// Mitsubishi GX Works2 project: part1 - Copy   PLC: FX3G

// global labels: Global1
VAR_GLOBAL
  start AT X007 : BOOL;
  helpStart AT M0 : BOOL;
  end_day AT X010 : BOOL;
  help_light AT M1 : BOOL;
  TC_200 AT TC200 : BOOL;
END_VAR
VAR_GLOBAL CONSTANT
  TIMER_1 : INT := 300;
END_VAR
VAR_GLOBAL
  TS_200 AT TS200 : BOOL;
  help_light2 AT M2 : BOOL;
  if_enough_stock AT M3 : BOOL;
  day_off AT M4 : BOOL;
END_VAR
VAR_GLOBAL CONSTANT
  zero : INT;
END_VAR
VAR_GLOBAL
  Cream AT D1100 : INT;
  cream_stock : INT;
  Chocolate AT D1101 : INT;
  chocolate_stock AT D1102 : INT;
  biscuit AT D1103 : INT;
  biscuit_stock AT D1104 : INT;
  start_Ziluf AT X011 : BOOL;
END_VAR
VAR_GLOBAL CONSTANT
  Cream300 : INT := 300;
END_VAR
VAR_GLOBAL
  ziluf_container AT D1105 : INT;
END_VAR
VAR_GLOBAL CONSTANT
  biscuit6 : INT := 6;
END_VAR
VAR_GLOBAL
  machineA AT X010 : BOOL;
  sen_mishtah AT X001 : BOOL;
  sen_camera AT X002 : BOOL;
  stop_machineA AT X005 : BOOL;
  sen_temp30 AT X003 : BOOL;
  sen_temp15 AT X004 : BOOL;
  ziluf_on AT Y004 : BOOL;
  finish_ziluf AT Y000 : BOOL;
  start_day AT Y007 : BOOL;
  m_5 AT M5 : BOOL;
  m_6 AT M6 : BOOL;
  m_7 AT M7 : BOOL;
  y_0 AT Y000 : BOOL;
  y_1 AT Y001 : BOOL;
  TS_1 AT TS1 : BOOL;
  m_0 AT M0 : BOOL;
  m_8 AT M8 : BOOL;
  TC_1 AT TC1 : BOOL;
END_VAR
VAR_GLOBAL CONSTANT
  sec_40 : INT := 40;
END_VAR
VAR_GLOBAL
  TC_2 AT TC2 : BOOL;
END_VAR
VAR_GLOBAL CONSTANT
  sec_1 : INT := 10;
END_VAR
VAR_GLOBAL
  TS_2 AT TS2 : BOOL;
  TC_3 AT TC3 : BOOL;
  TS_3 AT TS3 : BOOL;
  start_machineB AT X006 : BOOL;
END_VAR
VAR_GLOBAL CONSTANT
  div_400 : INT := 400;
END_VAR
VAR_GLOBAL
  analog_value : INT;
  m_9 AT M9 : BOOL;
END_VAR
VAR_GLOBAL CONSTANT
  Con : INT;
  Con0 : INT := 5;
  Con5 : INT := 5;
  CoN10 : INT := 10;
END_VAR
VAR_GLOBAL
  double_top AT M10 : BOOL;
END_VAR
VAR_GLOBAL CONSTANT
  Con6 : INT := 6;
END_VAR
VAR_GLOBAL
  regular_top AT M11 : BOOL;
  outRange AT M12 : BOOL;
  dip_container AT D1106 : INT;
END_VAR
VAR_GLOBAL CONSTANT
  Chocloate120 : INT := 120;
  Chocloate240 : INT := 240;
END_VAR
VAR_GLOBAL
  TC_4 AT TC4 : BOOL;
END_VAR
VAR_GLOBAL CONSTANT
  sec5 : INT := 50;
END_VAR
VAR_GLOBAL
  end_dip AT Y003 : BOOL;
  analog_input1 AT D8280 : INT;
  Analogvalue_result : BOOL;
  GT_result : REAL;
  TC_5 AT TC5 : BOOL;
END_VAR
VAR_GLOBAL CONSTANT
  sec_4 : INT := 40;
END_VAR
VAR_GLOBAL
  TS_5 AT TS5 : BOOL;
  y_3 AT Y003 : BOOL;
  finish_top AT M13 : BOOL;
  finish_regulartop AT M13 : BOOL;
  finish_doubletop AT M14 : BOOL;
  start_ariza AT X000 : BOOL;
  CC_1 AT CC1 : BOOL;
END_VAR
VAR_GLOBAL CONSTANT
  X0_value5 : INT := 5;
END_VAR
VAR_GLOBAL
  sof_ariza : BOOL;
  ariza AT X000 : BOOL;
  CC_2 AT CC2 : BOOL;
END_VAR
VAR_GLOBAL CONSTANT
  X0_value6 : INT := 6;
END_VAR
VAR_GLOBAL
  CS_1 AT CS1 : BOOL;
  CS_2 AT CS2 : BOOL;
  y_2 AT Y002 : BOOL;
  machineAhelp AT M15 : BOOL;
  end_prep AT M16 : BOOL;
  finish_prep AT M16 : BOOL;
  finish_iteration AT M17 : BOOL;
END_VAR
VAR_GLOBAL CONSTANT
  amount_6 : INT := 6;
END_VAR
VAR_GLOBAL
  total_krembo : INT;
  Check_stock AT M18 : BOOL;
END_VAR
VAR_GLOBAL CONSTANT
  min_6 : INT;
  min_300 : INT := 300;
  min_240 : INT := 240;
END_VAR
VAR_GLOBAL
  analog_output AT D8282 : INT;
END_VAR
VAR_GLOBAL CONSTANT
  Con_40 : INT := 40;
END_VAR
VAR_GLOBAL
  output_value : INT;
  if_enough_buiscit AT M19 : BOOL;
  if_enough_cream AT M20 : BOOL;
  if_enough_chocolate AT M21 : BOOL;
  TC_6 AT TC6 : BOOL;
  M_22 AT M22 : BOOL;
  TS_6 AT TS6 : BOOL;
END_VAR
VAR_GLOBAL CONSTANT
  sec_05 : INT := 5;
END_VAR
VAR_GLOBAL
  TC_7 AT TC7 : BOOL;
  TS_7 AT TS7 : BOOL;
  stock_ok AT M23 : BOOL;
  Check_first_stock AT M24 : BOOL;
  finish_fillstock AT M25 : BOOL;
  TC_8 AT TC8 : BOOL;
  TS_8 AT TS8 : BOOL;
END_VAR
VAR_GLOBAL CONSTANT
  CoNST0 : INT;
END_VAR
VAR_GLOBAL
  help_start AT M27 : BOOL;
  toping_kind : INT;
END_VAR

// task Task_01 (event TRUE, interval 0, priority 31): POU_01

PROGRAM POU_01
(* structured ladder/FBD written out as ST: instructions are called as NAME(EN, inputs, outputs); _pN, _eN, _tN stand for wires *)
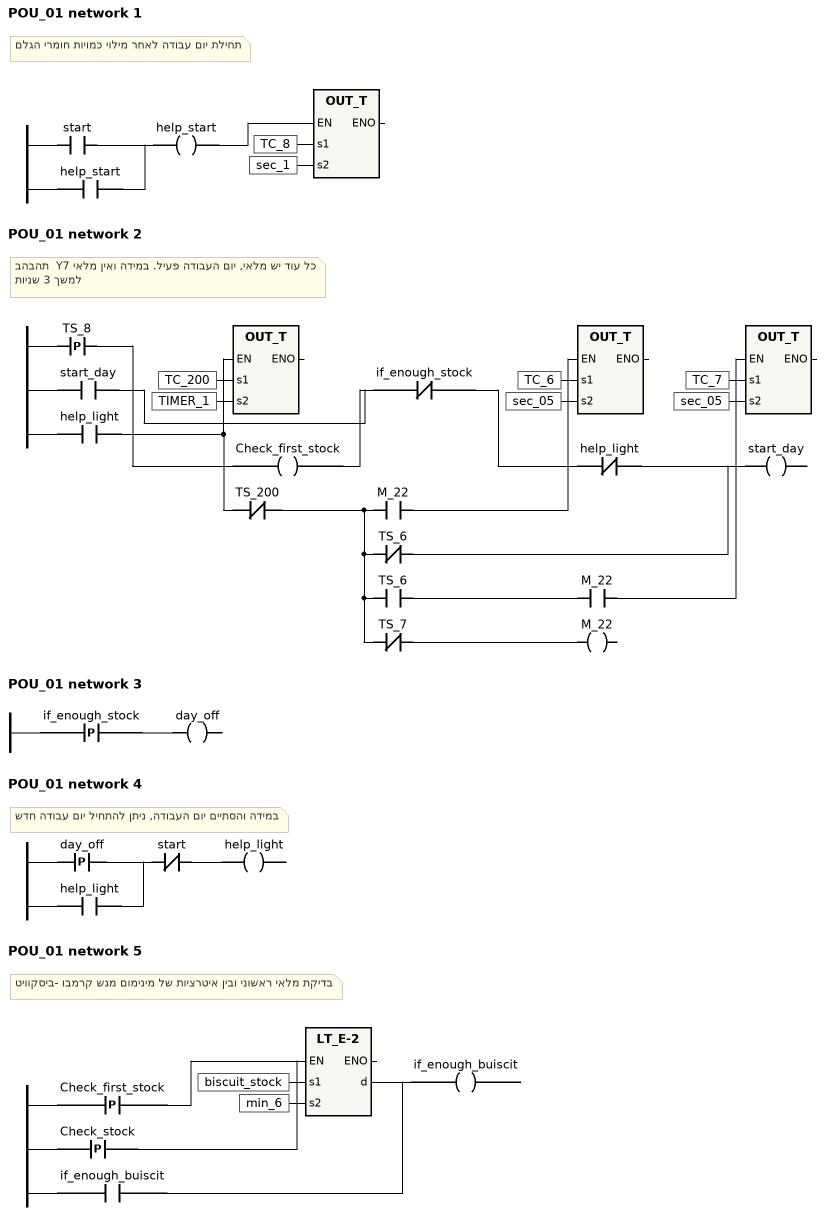
(* network 1 *)
(* תחילת יום עבודה לאחר מילוי כמויות חומרי הגלם *)
_p1 := start OR help_start;
help_start := _p1;
OUT_T(_p1, TC_8, sec_1);
(* network 2 *)
(* כל עוד יש מלאי, יום העבודה פעיל. במידה ואין מלאי Y7  תהבהב למשך 3 שניות *)
_p1 := LDP(TRUE, TS_8);
Check_first_stock := _p1;
_p2 := help_light AND NOT TS_200;
start_day := (((_p1 OR start_day) AND NOT if_enough_stock) AND NOT help_light) OR (_p2 AND NOT TS_6);
OUT_T(help_light, TC_200, TIMER_1);
OUT_T(_p2 AND M_22, TC_6, sec_05);
OUT_T(_p2 AND TS_6 AND M_22, TC_7, sec_05);
M_22 := _p2 AND NOT TS_7;
(* network 3 *)
day_off := LDP(TRUE, if_enough_stock);
(* network 4 *)
(* במידה והסתיים יום העבודה, ניתן להתחיל יום עבודה חדש *)
help_light := (LDP(TRUE, day_off) OR help_light) AND NOT start;
(* network 5 *)
(* בדיקת מלאי ראשוני ובין איטרציות של מינימום מגש קרמבו -ביסקוויט *)
LT_E(LDP(TRUE, Check_first_stock) OR LDP(TRUE, Check_stock), biscuit_stock, min_6, _t1);
if_enough_buiscit := _t1 OR if_enough_buiscit;
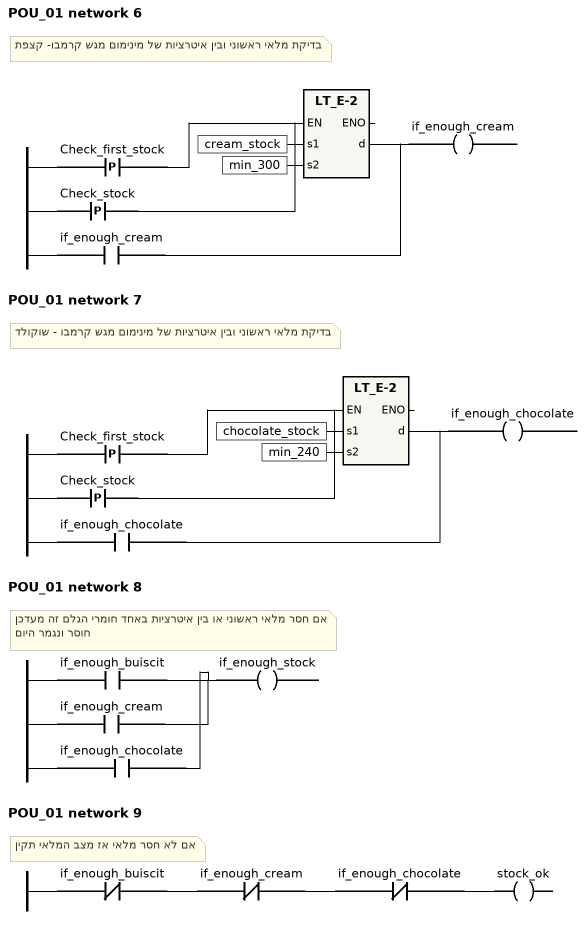
(* network 6 *)
(* בדיקת מלאי ראשוני ובין איטרציות של מינימום מגש קרמבו- קצפת *)
LT_E(LDP(TRUE, Check_first_stock) OR LDP(TRUE, Check_stock), cream_stock, min_300, _t1);
if_enough_cream := _t1 OR if_enough_cream;
(* network 7 *)
(* בדיקת מלאי ראשוני ובין איטרציות של מינימום מגש קרמבו - שוקולד *)
LT_E(LDP(TRUE, Check_first_stock) OR LDP(TRUE, Check_stock), chocolate_stock, min_240, _t1);
if_enough_chocolate := _t1 OR if_enough_chocolate;
(* network 8 *)
(* אם חסר מלאי ראשוני או בין איטרציות באחד חומרי הגלם זה מעדכן חוסר ונגמר היום *)
if_enough_stock := if_enough_buiscit OR if_enough_cream OR if_enough_chocolate;
(* network 9 *)
(* אם לא חסר מלאי אז מצב המלאי תקין *)
stock_ok := NOT if_enough_buiscit AND NOT if_enough_cream AND NOT if_enough_chocolate;
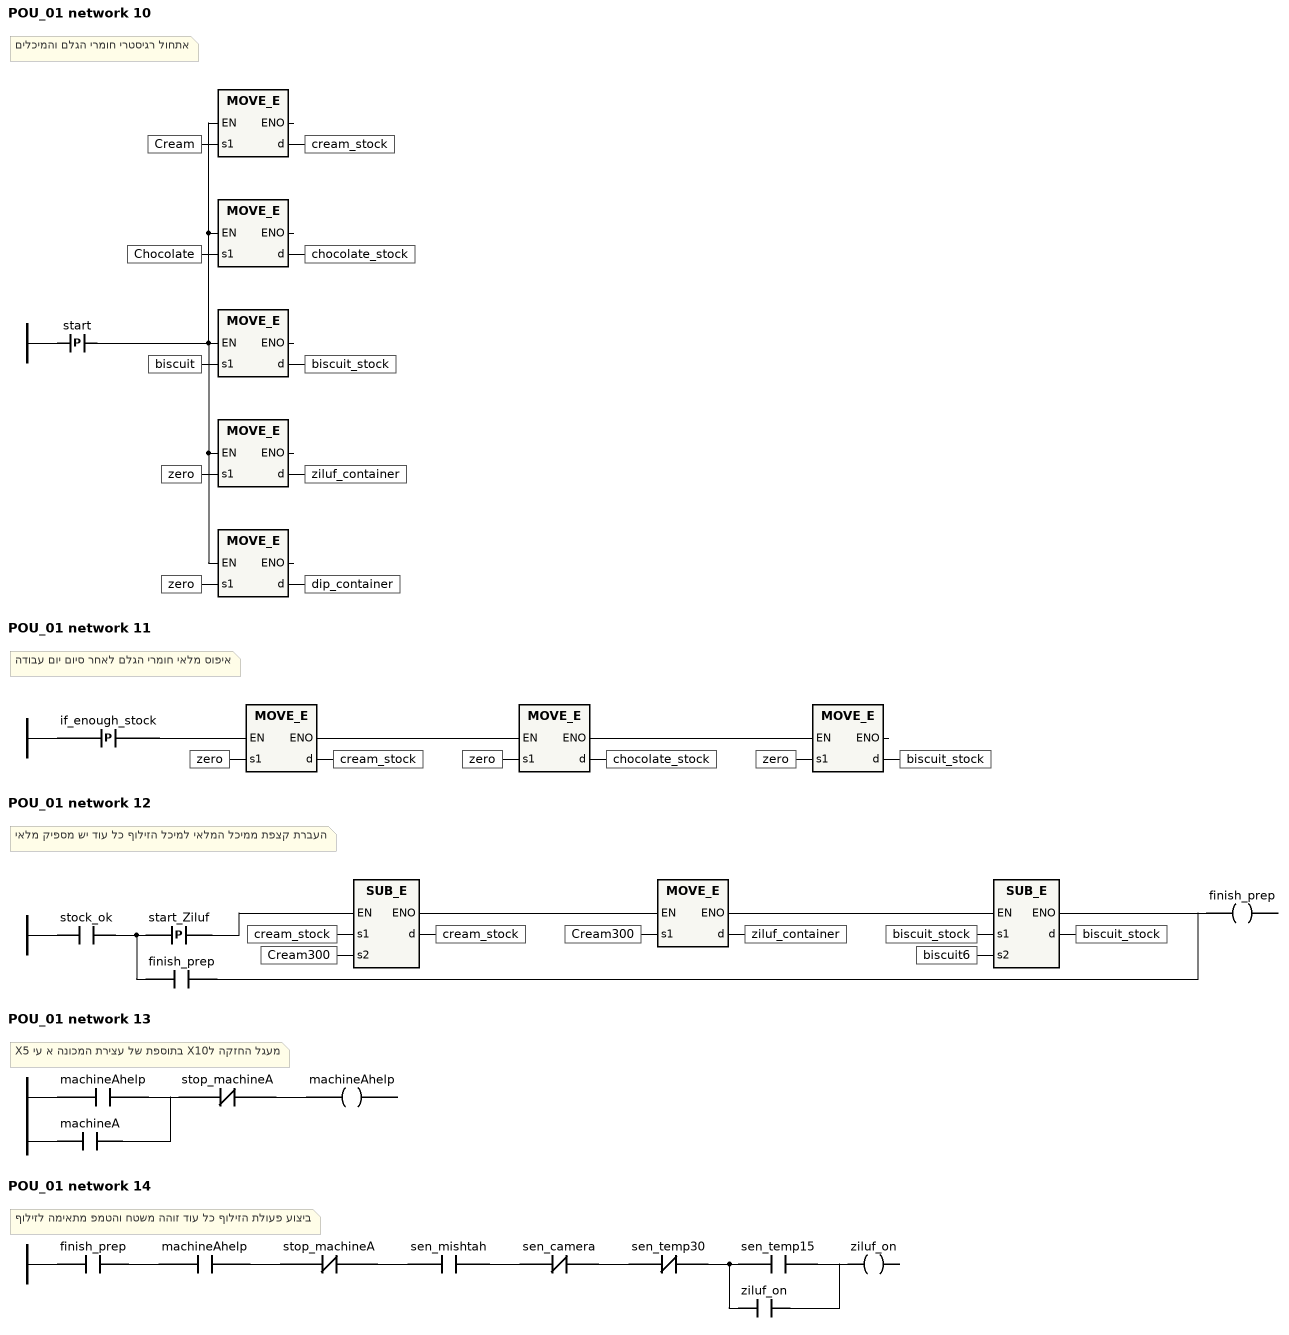
(* network 10 *)
(* אתחול רגיסטרי חומרי הגלם והמיכלים *)
_p1 := LDP(TRUE, start);
MOVE_E(_p1, Cream, cream_stock);
MOVE_E(_p1, Chocolate, chocolate_stock);
MOVE_E(_p1, biscuit, biscuit_stock);
MOVE_E(_p1, zero, ziluf_container);
MOVE_E(_p1, zero, dip_container);
(* network 11 *)
(* איפוס מלאי חומרי הגלם לאחר סיום יום עבודה *)
_e1 := MOVE_E(LDP(TRUE, if_enough_stock), zero, cream_stock);
_e2 := MOVE_E(_e1, zero, chocolate_stock);
MOVE_E(_e2, zero, biscuit_stock);
(* network 12 *)
(* העברת קצפת ממיכל המלאי למיכל הזילוף כל עוד יש מספיק מלאי *)
_e1 := SUB_E(stock_ok AND LDP(TRUE, start_Ziluf), cream_stock, Cream300, cream_stock);
_e2 := MOVE_E(_e1, Cream300, ziluf_container);
_e3 := SUB_E(_e2, biscuit_stock, biscuit6, biscuit_stock);
finish_prep := _e3 OR (stock_ok AND finish_prep);
(* network 13 *)
(* מעגל החזקה לX10 בתוספת של עצירת המכונה א עי X5 *)
machineAhelp := (machineAhelp OR machineA) AND NOT stop_machineA;
(* network 14 *)
(* ביצוע פעולת הזילוף כל עוד זוהה משטח והטמפ מתאימה לזילוף *)
_p1 := finish_prep AND machineAhelp AND NOT stop_machineA AND sen_mishtah AND NOT sen_camera AND NOT sen_temp30;
ziluf_on := (_p1 AND sen_temp15) OR (_p1 AND ziluf_on);
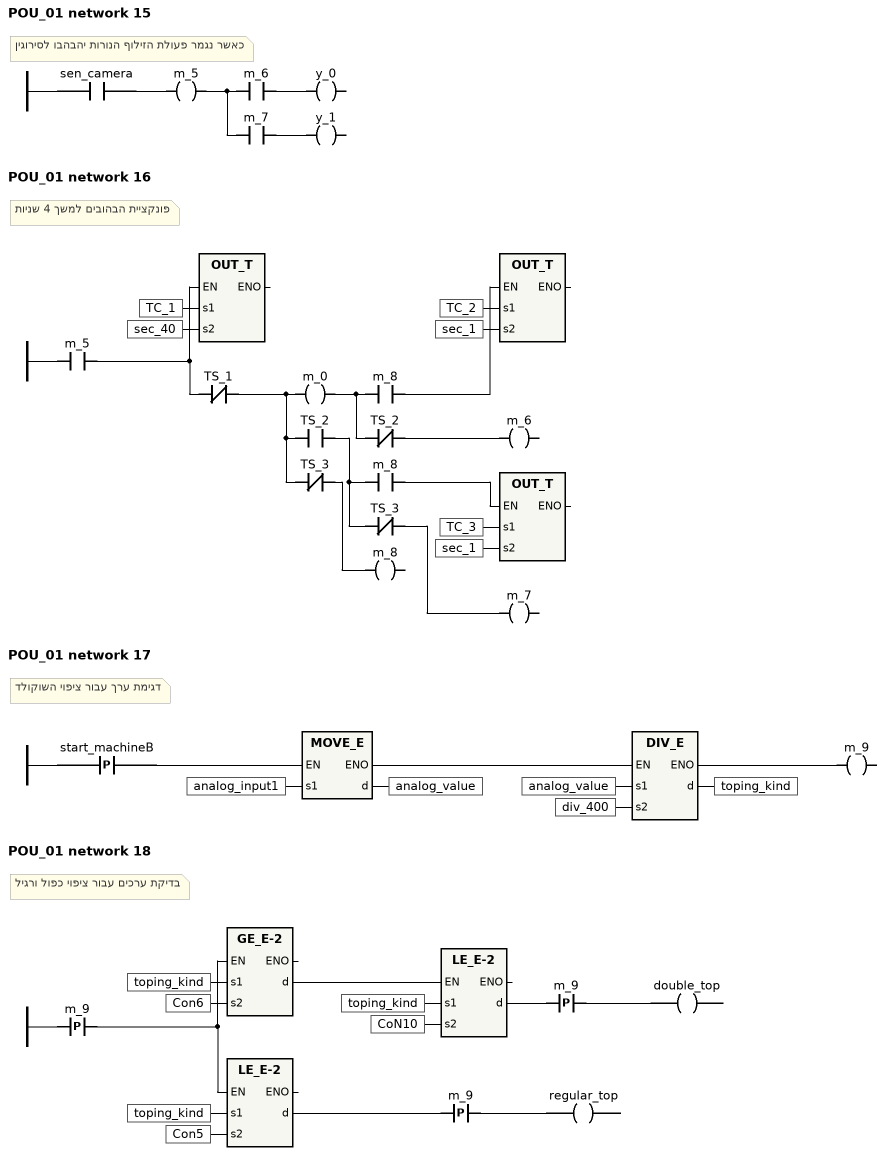
(* network 15 *)
(* כאשר נגמר פעולת הזילוף הנורות יהבהבו לסירוגין *)
m_5 := sen_camera;
y_0 := sen_camera AND m_6;
y_1 := sen_camera AND m_7;
(* network 16 *)
(* פונקציית הבהובים למשך 4 שניות *)
OUT_T(m_5, TC_1, sec_40);
_p1 := m_5 AND NOT TS_1;
m_0 := _p1;
OUT_T(_p1 AND m_8, TC_2, sec_1);
m_6 := _p1 AND NOT TS_2;
_p2 := _p1 AND TS_2;
OUT_T(_p2 AND m_8, TC_3, sec_1);
m_7 := _p2 AND NOT TS_3;
m_8 := _p1 AND NOT TS_3;
(* network 17 *)
(* דגימת ערך עבור ציפוי השוקולד *)
_e1 := MOVE_E(LDP(TRUE, start_machineB), analog_input1, analog_value);
_e2 := DIV_E(_e1, analog_value, div_400, toping_kind);
m_9 := _e2;
(* network 18 *)
(* בדיקת ערכים עבור ציפוי כפול ורגיל *)
_p1 := LDP(TRUE, m_9);
LE_E(_p1, toping_kind, Con5, _t2);
regular_top := _t2 AND LDP(TRUE, m_9);
GE_E(_p1, toping_kind, Con6, _t3);
LE_E(_t3, toping_kind, CoN10, _t4);
double_top := _t4 AND LDP(TRUE, m_9);
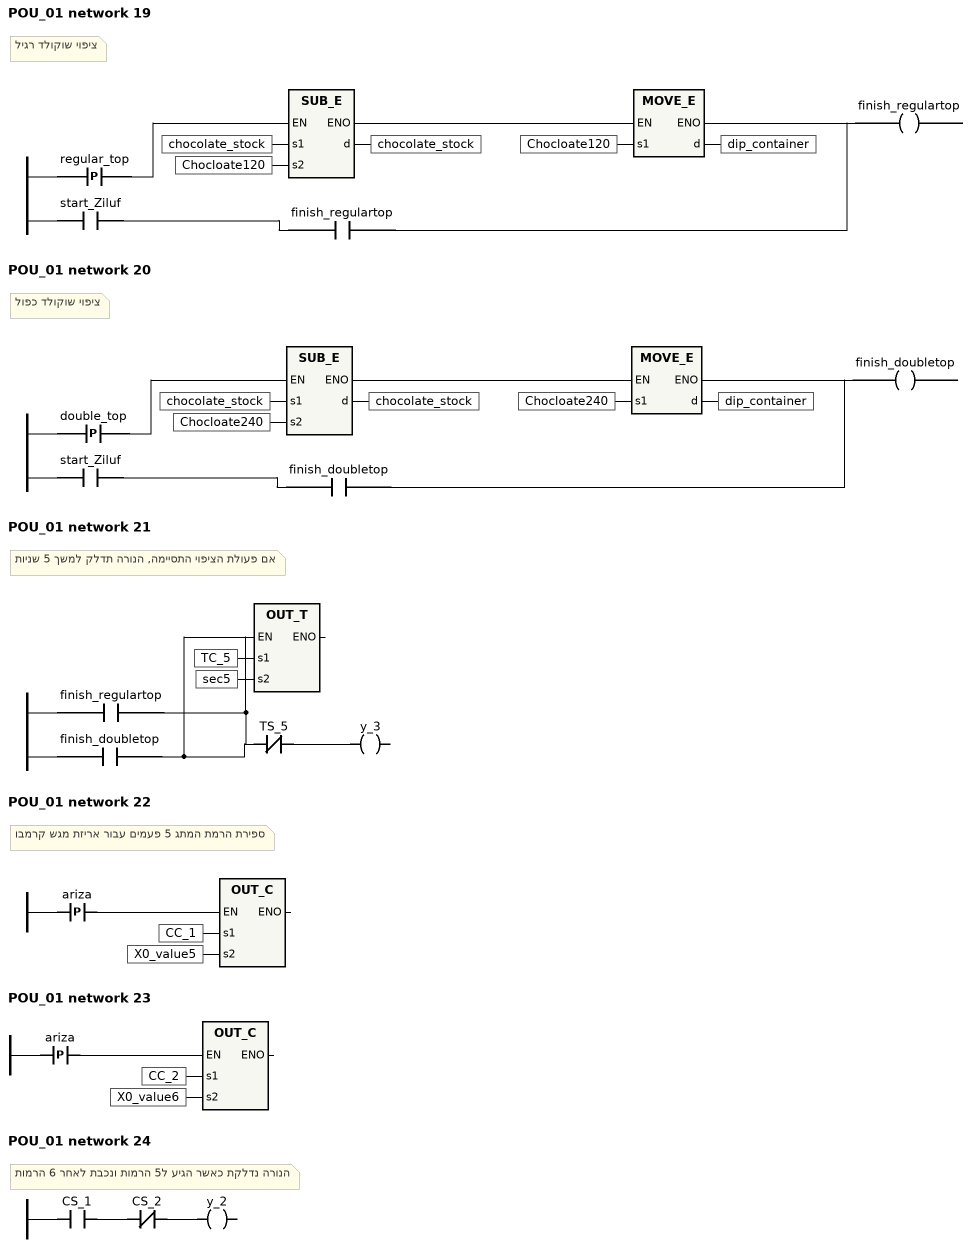
(* network 19 *)
(* ציפוי שוקולד רגיל *)
_e1 := SUB_E(LDP(TRUE, regular_top), chocolate_stock, Chocloate120, chocolate_stock);
_e2 := MOVE_E(_e1, Chocloate120, dip_container);
finish_regulartop := _e2 OR (start_Ziluf AND finish_regulartop);
(* network 20 *)
(* ציפוי שוקולד כפול *)
_e1 := SUB_E(LDP(TRUE, double_top), chocolate_stock, Chocloate240, chocolate_stock);
_e2 := MOVE_E(_e1, Chocloate240, dip_container);
finish_doubletop := _e2 OR (start_Ziluf AND finish_doubletop);
(* network 21 *)
(* אם פעולת הציפוי התסיימה, הנורה תדלק למשך 5 שניות *)
_p1 := finish_regulartop OR finish_doubletop;
OUT_T(_p1, TC_5, sec5);
y_3 := _p1 AND NOT TS_5;
(* network 22 *)
(* ספירת הרמת המתג 5 פעמים עבור אריזת מגש קרמבו *)
OUT_C(LDP(TRUE, ariza), CC_1, X0_value5);
(* network 23 *)
OUT_C(LDP(TRUE, ariza), CC_2, X0_value6);
(* network 24 *)
(* הנורה נדלקת כאשר הגיע ל5 הרמות ונכבת לאחר 6 הרמות *)
y_2 := CS_1 AND NOT CS_2;
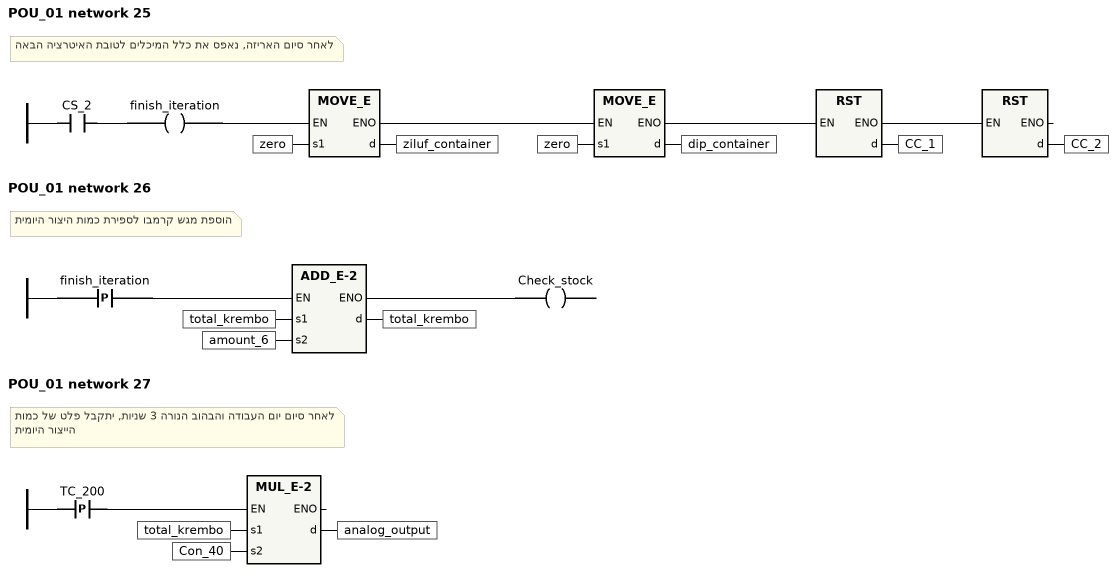
(* network 25 *)
(* לאחר סיום האריזה, נאפס את כלל המיכלים לטובת האיטרציה הבאה *)
finish_iteration := CS_2;
_e1 := MOVE_E(CS_2, zero, ziluf_container);
_e2 := MOVE_E(_e1, zero, dip_container);
_e3 := RST(_e2, CC_1);
RST(_e3, CC_2);
(* network 26 *)
(* הוספת מגש קרמבו לספירת כמות היצור היומית *)
_e1 := ADD_E(LDP(TRUE, finish_iteration), total_krembo, amount_6, total_krembo);
Check_stock := _e1;
(* network 27 *)
(* לאחר סיום יום העבודה והבהוב הנורה 3 שניות, יתקבל פלט של כמות הייצור היומית *)
MUL_E(LDP(TRUE, TC_200), total_krembo, Con_40, analog_output);
END_PROGRAM
